TYPE st_router_get :
STRUCT
	Device 		: 	st_Device;
	GPS			:	st_GPS;
	Mobile		:	st_mobile;
	Wifi		:	st_Wifi;
	e_SMSStatus : 	eSMSStatus;
	Events		:	st_Router_Events;
END_STRUCT
END_TYPE

(* stored: Version 1.1.0.1, ProductVersion 3.1.4026.18
   DUT st_router_get: Id {acfc0de7-5474-49bd-b092-b098fdfbac71} *)
